# B&R Automation Studio project HISTest (part 7)

#### HMI_Alarm.st
```iecst
ACTION ActTimeSplit:
	(**********************************************************************************)
	(* TIME TRANS 'DT#YYYY-MM-DD-hh:mm:ss' >> 'YY-MM-DD, hh:mm' *)
	(**********************************************************************************)
	Timestamp.DTGetTime_0();

	Timestamp.Original := DT_TO_STRING(Timestamp.DTGetTime_0.DT1);
	Timestamp.Split.Day := MID(Timestamp.Original,8,6);
	Timestamp.Split.Time := MID(Timestamp.Original,5,15);

	Timestamp.Total := CONCAT(Timestamp.Split.Day, CONCAT(', ',Timestamp.Split.Time));
END_ACTION
ACTION ActSystem_Warning:

	IF EDGEPOS(PMS.SysBatProtect.Field.BSA_Alarm_OC) THEN
		IF HMI_Alarm.Warning[0].Count = 0 THEN
			HMI_Alarm.Warning[0].InitialTime 	:= Timestamp.Total;
			HMI_Alarm.Warning[0].RecentTime 	:= Timestamp.Total;
		ELSE
			HMI_Alarm.Warning[0].RecentTime 	:= Timestamp.Total;
		END_IF;
		HMI_Alarm.Warning[0].Count  := HMI_Alarm.Warning[0].Count + 1;
	END_IF;
	IF EDGEPOS(PMS.SysBatProtect.Field.BSA_Alarm_SOC_OV) THEN
		IF HMI_Alarm.Warning[1].Count = 0 THEN
			HMI_Alarm.Warning[1].InitialTime  	:= Timestamp.Total;
			HMI_Alarm.Warning[1].RecentTime 	:= Timestamp.Total;
		ELSE
			HMI_Alarm.Warning[1].InitialTime  	:= Timestamp.Total;
		END_IF;
		HMI_Alarm.Warning[1].Count  := HMI_Alarm.Warning[1].Count + 1;
	END_IF;
	IF EDGEPOS(PMS.SysBatProtect.Field.BSA_Alarm_SOC_UN) THEN
		IF HMI_Alarm.Warning[2].Count = 0 THEN
			HMI_Alarm.Warning[2].InitialTime  	:= Timestamp.Total;
			HMI_Alarm.Warning[2].RecentTime 	:= Timestamp.Total;
		ELSE
			HMI_Alarm.Warning[2].InitialTime  	:= Timestamp.Total;
		END_IF;
		HMI_Alarm.Warning[2].Count  := HMI_Alarm.Warning[2].Count + 1;
	END_IF;
	IF EDGEPOS(PMS.SysBatProtect.Field.BSA_Alarm_OV) THEN
		IF HMI_Alarm.Warning[3].Count = 0 THEN
			HMI_Alarm.Warning[3].InitialTime  	:= Timestamp.Total;
			HMI_Alarm.Warning[3].RecentTime 	:= Timestamp.Total;
		ELSE
			HMI_Alarm.Warning[3].InitialTime  	:= Timestamp.Total;
		END_IF;
		HMI_Alarm.Warning[3].Count  := HMI_Alarm.Warning[3].Count + 1;
	END_IF;
	IF EDGEPOS(PMS.SysBatProtect.Field.BSA_Alarm_UV) THEN
		IF HMI_Alarm.Warning[4].Count = 0 THEN
			HMI_Alarm.Warning[4].InitialTime  	:= Timestamp.Total;
			HMI_Alarm.Warning[4].RecentTime 	:= Timestamp.Total;
		ELSE
			HMI_Alarm.Warning[4].InitialTime  	:= Timestamp.Total;
		END_IF;
		HMI_Alarm.Warning[4].Count  := HMI_Alarm.Warning[4].Count + 1;
	END_IF;
	IF EDGEPOS(PMS.SysBatProtect.Field.BSA_Alarm_Cell_OV) THEN
		IF HMI_Alarm.Warning[5].Count = 0 THEN
			HMI_Alarm.Warning[5].InitialTime  	:= Timestamp.Total;
			HMI_Alarm.Warning[5].RecentTime 	:= Timestamp.Total;
		ELSE
			HMI_Alarm.Warning[5].InitialTime  	:= Timestamp.Total;
		END_IF;
		HMI_Alarm.Warning[5].Count  := HMI_Alarm.Warning[5].Count + 1;
	END_IF;
	IF EDGEPOS(PMS.SysBatProtect.Field.BSA_Alarm_Cell_UV) THEN
		IF HMI_Alarm.Warning[6].Count = 0 THEN
			HMI_Alarm.Warning[6].InitialTime  	:= Timestamp.Total;
			HMI_Alarm.Warning[6].RecentTime 	:= Timestamp.Total;
		ELSE
			HMI_Alarm.Warning[6].InitialTime  	:= Timestamp.Total;
		END_IF;
		HMI_Alarm.Warning[6].Count  := HMI_Alarm.Warning[6].Count + 1;
	END_IF;
	IF EDGEPOS(PMS.SysBatProtect.Field.BSA_Alarm_Cell_UnBalaV) THEN
		IF HMI_Alarm.Warning[7].Count = 0 THEN
			HMI_Alarm.Warning[7].InitialTime  	:= Timestamp.Total;
			HMI_Alarm.Warning[7].RecentTime 	:= Timestamp.Total;
		ELSE
			HMI_Alarm.Warning[7].InitialTime  	:= Timestamp.Total;
		END_IF;
		HMI_Alarm.Warning[7].Count  := HMI_Alarm.Warning[7].Count + 1;
	END_IF;
	IF EDGEPOS(PMS.SysBatProtect.Field.BSA_Alarm_Discharger_Cell_OT) THEN
		IF HMI_Alarm.Warning[8].Count = 0 THEN
			HMI_Alarm.Warning[8].InitialTime  	:= Timestamp.Total;
			HMI_Alarm.Warning[8].RecentTime 	:= Timestamp.Total;
		ELSE
			HMI_Alarm.Warning[8].InitialTime  	:= Timestamp.Total;
		END_IF;
		HMI_Alarm.Warning[8].Count  := HMI_Alarm.Warning[8].Count + 1;
	END_IF;
	IF EDGEPOS(PMS.SysBatProtect.Field.BSA_Alarm_Charger_Cell_OT) THEN
		IF HMI_Alarm.Warning[9].Count = 0 THEN
			HMI_Alarm.Warning[9].InitialTime  	:= Timestamp.Total;
			HMI_Alarm.Warning[9].RecentTime 	:= Timestamp.Total;
		ELSE
			HMI_Alarm.Warning[9].InitialTime  	:= Timestamp.Total;
		END_IF;
		HMI_Alarm.Warning[9].Count  := HMI_Alarm.Warning[9].Count + 1;
	END_IF;
	IF EDGEPOS(PMS.SysBatProtect.Field.BSA_Alarm_Discharger_Cell_UT) THEN
		IF HMI_Alarm.Warning[10].Count = 0 THEN
			HMI_Alarm.Warning[10].InitialTime  	:= Timestamp.Total;
			HMI_Alarm.Warning[10].RecentTime 	:= Timestamp.Total;
		ELSE
			HMI_Alarm.Warning[10].InitialTime  	:= Timestamp.Total;
		END_IF;
		HMI_Alarm.Warning[10].Count 	:= HMI_Alarm.Warning[10].Count + 1;
	END_IF;
	IF EDGEPOS(PMS.SysBatProtect.Field.BSA_Alarm_Charger_Cell_UT) THEN
		IF HMI_Alarm.Warning[11].Count = 0 THEN
			HMI_Alarm.Warning[11].InitialTime  	:= Timestamp.Total;
			HMI_Alarm.Warning[11].RecentTime 	:= Timestamp.Total;
		ELSE
			HMI_Alarm.Warning[11].InitialTime  	:= Timestamp.Total;
		END_IF;
		HMI_Alarm.Warning[11].Count 	:= HMI_Alarm.Warning[11].Count + 1;
	END_IF;
	IF EDGEPOS(PMS.SysBatProtect.Field.BSA_Alarm_Cell_UnBalaT) THEN
		IF HMI_Alarm.Warning[12].Count = 0 THEN
			HMI_Alarm.Warning[12].InitialTime  	:= Timestamp.Total;
			HMI_Alarm.Warning[12].RecentTime 	:= Timestamp.Total;
		ELSE
			HMI_Alarm.Warning[12].InitialTime  	:= Timestamp.Total;
		END_IF;
		HMI_Alarm.Warning[12].Count 	:= HMI_Alarm.Warning[12].Count + 1;
	END_IF;

END_ACTION
ACTION ActSystem_Fault: //
	IF EDGEPOS(PMS.SysBatProtect.Field.BSA_Fault_OC) THEN
		IF HMI_Alarm.Fault[0].Count = 0 THEN
			HMI_Alarm.Fault[0].InitialTime 	:= Timestamp.Total;
			HMI_Alarm.Fault[0].RecentTime 	:= Timestamp.Total;
		ELSE
			HMI_Alarm.Fault[0].RecentTime 	:= Timestamp.Total;
		END_IF;
		HMI_Alarm.Fault[0].Count  := HMI_Alarm.Fault[0].Count + 1;
	END_IF;
	IF EDGEPOS(PMS.SysBatProtect.Field.BSA_Fault_SOC_OV) THEN
		IF HMI_Alarm.Fault[1].Count = 0 THEN
			HMI_Alarm.Fault[1].InitialTime  	:= Timestamp.Total;
			HMI_Alarm.Fault[1].RecentTime 	:= Timestamp.Total;
		ELSE
			HMI_Alarm.Fault[1].InitialTime  	:= Timestamp.Total;
		END_IF;
		HMI_Alarm.Fault[1].Count  := HMI_Alarm.Fault[1].Count + 1;
	END_IF;
	IF EDGEPOS(PMS.SysBatProtect.Field.BSA_Fault_SOC_UN) THEN
		IF HMI_Alarm.Fault[2].Count = 0 THEN
			HMI_Alarm.Fault[2].InitialTime  	:= Timestamp.Total;
			HMI_Alarm.Fault[2].RecentTime 	:= Timestamp.Total;
		ELSE
			HMI_Alarm.Fault[2].InitialTime  	:= Timestamp.Total;
		END_IF;
		HMI_Alarm.Fault[2].Count  := HMI_Alarm.Fault[2].Count + 1;
	END_IF;
	IF EDGEPOS(PMS.SysBatProtect.Field.BSA_Fault_OV) THEN
		IF HMI_Alarm.Fault[3].Count = 0 THEN
			HMI_Alarm.Fault[3].InitialTime  	:= Timestamp.Total;
			HMI_Alarm.Fault[3].RecentTime 	:= Timestamp.Total;
		ELSE
			HMI_Alarm.Fault[3].InitialTime  	:= Timestamp.Total;
		END_IF;
		HMI_Alarm.Fault[3].Count  := HMI_Alarm.Fault[3].Count + 1;
	END_IF;
	IF EDGEPOS(PMS.SysBatProtect.Field.BSA_Fault_UV) THEN
		IF HMI_Alarm.Fault[4].Count = 0 THEN
			HMI_Alarm.Fault[4].InitialTime  	:= Timestamp.Total;
			HMI_Alarm.Fault[4].RecentTime 	:= Timestamp.Total;
		ELSE
			HMI_Alarm.Fault[4].InitialTime  	:= Timestamp.Total;
		END_IF;
		HMI_Alarm.Fault[4].Count  := HMI_Alarm.Fault[4].Count + 1;
	END_IF;
	IF EDGEPOS(PMS.SysBatProtect.Field.BSA_Fault_Cell_OV) THEN
		IF HMI_Alarm.Fault[5].Count = 0 THEN
			HMI_Alarm.Fault[5].InitialTime  	:= Timestamp.Total;
			HMI_Alarm.Fault[5].RecentTime 	:= Timestamp.Total;
		ELSE
			HMI_Alarm.Fault[5].InitialTime  	:= Timestamp.Total;
		END_IF;
		HMI_Alarm.Fault[5].Count  := HMI_Alarm.Fault[5].Count + 1;
	END_IF;
	IF EDGEPOS(PMS.SysBatProtect.Field.BSA_Fault_Cell_UV) THEN
		IF HMI_Alarm.Fault[6].Count = 0 THEN
			HMI_Alarm.Fault[6].InitialTime  	:= Timestamp.Total;
			HMI_Alarm.Fault[6].RecentTime 	:= Timestamp.Total;
		ELSE
			HMI_Alarm.Fault[6].InitialTime  	:= Timestamp.Total;
		END_IF;
		HMI_Alarm.Fault[6].Count  := HMI_Alarm.Fault[6].Count + 1;
	END_IF;
	IF EDGEPOS(PMS.SysBatProtect.Field.BSA_Fault_Cell_UnBalaV) THEN
		IF HMI_Alarm.Fault[7].Count = 0 THEN
			HMI_Alarm.Fault[7].InitialTime  	:= Timestamp.Total;
			HMI_Alarm.Fault[7].RecentTime 	:= Timestamp.Total;
		ELSE
			HMI_Alarm.Fault[7].InitialTime  	:= Timestamp.Total;
		END_IF;
		HMI_Alarm.Fault[7].Count  := HMI_Alarm.Fault[7].Count + 1;
	END_IF;
	IF EDGEPOS(PMS.SysBatProtect.Field.BSA_Fault_Discharger_Cell_OT) THEN
		IF HMI_Alarm.Fault[8].Count = 0 THEN
			HMI_Alarm.Fault[8].InitialTime  	:= Timestamp.Total;
			HMI_Alarm.Fault[8].RecentTime 	:= Timestamp.Total;
		ELSE
			HMI_Alarm.Fault[8].InitialTime  	:= Timestamp.Total;
		END_IF;
		HMI_Alarm.Fault[8].Count  := HMI_Alarm.Fault[8].Count + 1;
	END_IF;
	IF EDGEPOS(PMS.SysBatProtect.Field.BSA_Fault_Charger_Cell_OT) THEN
		IF HMI_Alarm.Fault[9].Count = 0 THEN
			HMI_Alarm.Fault[9].InitialTime  	:= Timestamp.Total;
			HMI_Alarm.Fault[9].RecentTime 	:= Timestamp.Total;
		ELSE
			HMI_Alarm.Fault[9].InitialTime  	:= Timestamp.Total;
		END_IF;
		HMI_Alarm.Fault[9].Count  := HMI_Alarm.Fault[9].Count + 1;
	END_IF;
	IF EDGEPOS(PMS.SysBatProtect.Field.BSA_Fault_Discharger_Cell_UT) THEN
		IF HMI_Alarm.Fault[10].Count = 0 THEN
			HMI_Alarm.Fault[10].InitialTime  	:= Timestamp.Total;
			HMI_Alarm.Fault[10].RecentTime 	:= Timestamp.Total;
		ELSE
			HMI_Alarm.Fault[10].InitialTime  	:= Timestamp.Total;
		END_IF;
		HMI_Alarm.Fault[10].Count 	:= HMI_Alarm.Fault[10].Count + 1;
	END_IF;
	IF EDGEPOS(PMS.SysBatProtect.Field.BSA_Fault_Charger_Cell_UT) THEN
		IF HMI_Alarm.Fault[11].Count = 0 THEN
			HMI_Alarm.Fault[11].InitialTime  	:= Timestamp.Total;
			HMI_Alarm.Fault[11].RecentTime 	:= Timestamp.Total;
		ELSE
			HMI_Alarm.Fault[11].InitialTime  	:= Timestamp.Total;
		END_IF;
		HMI_Alarm.Fault[11].Count 	:= HMI_Alarm.Fault[11].Count + 1;
	END_IF;
	IF EDGEPOS(PMS.SysBatProtect.Field.BSA_Fault_Cell_UnBalaT) THEN
		IF HMI_Alarm.Fault[12].Count = 0 THEN
			HMI_Alarm.Fault[12].InitialTime  	:= Timestamp.Total;
			HMI_Alarm.Fault[12].RecentTime 	:= Timestamp.Total;
		ELSE
			HMI_Alarm.Fault[12].InitialTime  	:= Timestamp.Total;
		END_IF;
		HMI_Alarm.Fault[12].Count 	:= HMI_Alarm.Fault[12].Count + 1;
	END_IF;
END_ACTION
ACTION ActSystem_Protect:

	IF EDGEPOS(PMS.SysBatProtect.Field.BSA_Prtct_OC) THEN

		IF HMI_Alarm.Protect[0].Count = 0 THEN
			HMI_Alarm.Protect[0].InitialTime 	:= Timestamp.Total;
			HMI_Alarm.Protect[0].RecentTime 	:= Timestamp.Total;
		ELSE
			HMI_Alarm.Protect[0].RecentTime 	:= Timestamp.Total;
		END_IF;
		HMI_Alarm.Protect[0].Count  := HMI_Alarm.Protect[0].Count + 1;
	END_IF;
	IF EDGEPOS(PMS.SysBatProtect.Field.BSA_Prtct_SOC_OV) THEN

		IF HMI_Alarm.Protect[1].Count = 0 THEN
			HMI_Alarm.Protect[1].InitialTime  	:= Timestamp.Total;
			HMI_Alarm.Protect[1].RecentTime 	:= Timestamp.Total;
		ELSE
			HMI_Alarm.Protect[1].RecentTime  	:= Timestamp.Total;
		END_IF;
		HMI_Alarm.Protect[1].Count  := HMI_Alarm.Protect[1].Count + 1;
	END_IF;
	IF EDGEPOS(PMS.SysBatProtect.Field.BSA_Prtct_SOC_UN) THEN

		IF HMI_Alarm.Protect[2].Count = 0 THEN
			HMI_Alarm.Protect[2].InitialTime  	:= Timestamp.Total;
			HMI_Alarm.Protect[2].RecentTime 	:= Timestamp.Total;
		ELSE
			HMI_Alarm.Protect[2].RecentTime  	:= Timestamp.Total;
		END_IF;
		HMI_Alarm.Protect[2].Count  := HMI_Alarm.Protect[2].Count + 1;
	END_IF;
	IF EDGEPOS(PMS.SysBatProtect.Field.BSA_Prtct_OV) THEN

		IF HMI_Alarm.Protect[3].Count = 0 THEN
			HMI_Alarm.Protect[3].InitialTime  	:= Timestamp.Total;
			HMI_Alarm.Protect[3].RecentTime 	:= Timestamp.Total;
		ELSE
			HMI_Alarm.Protect[3].RecentTime  	:= Timestamp.Total;
		END_IF;
		HMI_Alarm.Protect[3].Count  := HMI_Alarm.Protect[3].Count + 1;
	END_IF;
	IF EDGEPOS(PMS.SysBatProtect.Field.BSA_Prtct_UV) THEN

		IF HMI_Alarm.Protect[4].Count = 0 THEN
			HMI_Alarm.Protect[4].InitialTime  	:= Timestamp.Total;
			HMI_Alarm.Protect[4].RecentTime 	:= Timestamp.Total;
		ELSE
			HMI_Alarm.Protect[4].RecentTime  	:= Timestamp.Total;
		END_IF;
		HMI_Alarm.Protect[4].Count  := HMI_Alarm.Protect[4].Count + 1;
	END_IF;
	IF EDGEPOS(PMS.SysBatProtect.Field.BSA_Prtct_Cell_OV) THEN

		IF HMI_Alarm.Protect[5].Count = 0 THEN
			HMI_Alarm.Protect[5].InitialTime  	:= Timestamp.Total;
			HMI_Alarm.Protect[5].RecentTime 	:= Timestamp.Total;
		ELSE
			HMI_Alarm.Protect[5].RecentTime  	:= Timestamp.Total;
		END_IF;
		HMI_Alarm.Protect[5].Count  := HMI_Alarm.Protect[5].Count + 1;
	END_IF;
	IF EDGEPOS(PMS.SysBatProtect.Field.BSA_Prtct_Cell_UV) THEN

		IF HMI_Alarm.Protect[6].Count = 0 THEN
			HMI_Alarm.Protect[6].InitialTime  	:= Timestamp.Total;
			HMI_Alarm.Protect[6].RecentTime 	:= Timestamp.Total;
		ELSE
			HMI_Alarm.Protect[6].RecentTime  	:= Timestamp.Total;
		END_IF;
		HMI_Alarm.Protect[6].Count  := HMI_Alarm.Protect[6].Count + 1;
	END_IF;
	IF EDGEPOS(PMS.SysBatProtect.Field.BSA_Prtct_Cell_UnBalaV) THEN

		IF HMI_Alarm.Protect[7].Count = 0 THEN
			HMI_Alarm.Protect[7].InitialTime  	:= Timestamp.Total;
			HMI_Alarm.Protect[7].RecentTime 	:= Timestamp.Total;
		ELSE
			HMI_Alarm.Protect[7].RecentTime  	:= Timestamp.Total;
		END_IF;
		HMI_Alarm.Protect[7].Count  := HMI_Alarm.Protect[7].Count + 1;
	END_IF;
	IF EDGEPOS(PMS.SysBatProtect.Field.BSA_Prtct_Discharger_Cell_OT) THEN

		IF HMI_Alarm.Protect[8].Count = 0 THEN
			HMI_Alarm.Protect[8].InitialTime  	:= Timestamp.Total;
			HMI_Alarm.Protect[8].RecentTime 	:= Timestamp.Total;
		ELSE
			HMI_Alarm.Protect[8].RecentTime  	:= Timestamp.Total;
		END_IF;
		HMI_Alarm.Protect[8].Count  := HMI_Alarm.Protect[8].Count + 1;
	END_IF;
	IF EDGEPOS(PMS.SysBatProtect.Field.BSA_Prtct_Charger_Cell_OT) THEN

		IF HMI_Alarm.Protect[9].Count = 0 THEN
			HMI_Alarm.Protect[9].InitialTime  	:= Timestamp.Total;
			HMI_Alarm.Protect[9].RecentTime 	:= Timestamp.Total;
		ELSE
			HMI_Alarm.Protect[9].RecentTime  	:= Timestamp.Total;
		END_IF;
		HMI_Alarm.Protect[9].Count  := HMI_Alarm.Protect[9].Count + 1;
	END_IF;
	IF EDGEPOS(PMS.SysBatProtect.Field.BSA_Prtct_Discharger_Cell_UT) THEN

		IF HMI_Alarm.Protect[10].Count = 0 THEN
			HMI_Alarm.Protect[10].InitialTime  	:= Timestamp.Total;
			HMI_Alarm.Protect[10].RecentTime 	:= Timestamp.Total;
		ELSE
			HMI_Alarm.Protect[10].RecentTime  	:= Timestamp.Total;
		END_IF;
		HMI_Alarm.Protect[10].Count 	:= HMI_Alarm.Protect[10].Count + 1;
	END_IF;
	IF EDGEPOS(PMS.SysBatProtect.Field.BSA_Prtct_Charger_Cell_UT) THEN

		IF HMI_Alarm.Protect[11].Count = 0 THEN
			HMI_Alarm.Protect[11].InitialTime  	:= Timestamp.Total;
			HMI_Alarm.Protect[11].RecentTime 	:= Timestamp.Total;
		ELSE
			HMI_Alarm.Protect[11].RecentTime  	:= Timestamp.Total;
		END_IF;
		HMI_Alarm.Protect[11].Count 	:= HMI_Alarm.Protect[11].Count + 1;
	END_IF;
	IF EDGEPOS(PMS.SysBatProtect.Field.BSA_Prtct_Cell_UnBalaT) THEN

		IF HMI_Alarm.Protect[12].Count = 0 THEN
			HMI_Alarm.Protect[12].InitialTime  	:= Timestamp.Total;
			HMI_Alarm.Protect[12].RecentTime 	:= Timestamp.Total;
		ELSE
			HMI_Alarm.Protect[12].RecentTime  	:= Timestamp.Total;
		END_IF;
		HMI_Alarm.Protect[12].Count 	:= HMI_Alarm.Protect[12].Count + 1;
	END_IF;
	IF EDGEPOS(PMS.SysBatProtect.Field.BSA_Prtct_RelayWelding) THEN

		IF HMI_Alarm.Protect[13].Count = 0 THEN
			HMI_Alarm.Protect[13].InitialTime  	:= Timestamp.Total;
			HMI_Alarm.Protect[13].RecentTime 	:= Timestamp.Total;
		ELSE
			HMI_Alarm.Protect[13].RecentTime  	:= Timestamp.Total;
		END_IF;
		HMI_Alarm.Protect[13].Count 	:= HMI_Alarm.Protect[13].Count + 1;
	END_IF;
	IF EDGEPOS(PMS.SysBatProtect.Field.BSA_Prtct_InternalCOM) THEN

		IF HMI_Alarm.Protect[14].Count = 0 THEN
			HMI_Alarm.Protect[14].InitialTime  	:= Timestamp.Total;
			HMI_Alarm.Protect[14].RecentTime 	:= Timestamp.Total;
		ELSE
			HMI_Alarm.Protect[14].RecentTime  	:= Timestamp.Total;
		END_IF;
		HMI_Alarm.Protect[14].Count 	:= HMI_Alarm.Protect[14].Count + 1;
	END_IF;
	IF EDGEPOS(PMS.SysBatProtect.Field.BSA_Prtct_ExternalCOM) THEN

		IF HMI_Alarm.Protect[15].Count = 0 THEN
			HMI_Alarm.Protect[15].InitialTime  	:= Timestamp.Total;
			HMI_Alarm.Protect[15].RecentTime 	:= Timestamp.Total;
		ELSE
			HMI_Alarm.Protect[15].RecentTime  	:= Timestamp.Total;
		END_IF;
		HMI_Alarm.Protect[15].Count 	:= HMI_Alarm.Protect[15].Count + 1;
	END_IF;
//	IF EDGEPOS(PMS.SysBatProtect.Field.BSA_Prtct_CT_COM_Err) THEN
//
//		IF HMI_Alarm.Protect[16].Count = 0 THEN
//			HMI_Alarm.Protect[16].InitialTime  	:= Timestamp.Total;
//			HMI_Alarm.Protect[16].RecentTime 	:= Timestamp.Total;
//		ELSE
//			HMI_Alarm.Protect[16].InitialTime  	:= Timestamp.Total;
//		END_IF;
//		HMI_Alarm.Protect[16].Count 	:= HMI_Alarm.Protect[16].Count + 1;
//	END_IF;
	IF EDGEPOS(PMS.SysBatProtect.Field.BSA_Prtct_WaterLeak) THEN

		IF HMI_Alarm.Protect[17].Count = 0 THEN
			HMI_Alarm.Protect[17].InitialTime  	:= Timestamp.Total;
			HMI_Alarm.Protect[17].RecentTime 	:= Timestamp.Total;
		ELSE
			HMI_Alarm.Protect[17].RecentTime  	:= Timestamp.Total;
		END_IF;
		HMI_Alarm.Protect[17].Count 	:= HMI_Alarm.Protect[17].Count + 1;
	END_IF;
//	IF EDGEPOS(PMS.SysBatProtect.Field.BSA_Prtct_EMS_SW_Err) THEN
//
//		IF HMI_Alarm.Protect[18].Count = 0 THEN
//			HMI_Alarm.Protect[18].InitialTime  	:= Timestamp.Total;
//			HMI_Alarm.Protect[18].RecentTime 	:= Timestamp.Total;
//		ELSE
//			HMI_Alarm.Protect[18].InitialTime  	:= Timestamp.Total;
//		END_IF;
//		HMI_Alarm.Protect[18].Count 	:= HMI_Alarm.Protect[18].Count + 1;
//	END_IF;

	IF NOT(HMI.DialogBox.Protect_Trigger) THEN
		FOR LoopNum := 0 TO 18 DO
			IF HMI_Alarm.Protect[LoopNum].Count > 0 THEN
				HMI.DialogBox.Protect_Trigger 	:= TRUE;
				HMI.DialogBox.ProtectName		:=	HMI_Alarm.Protect[LoopNum].Name;
				EXIT;
			END_IF;
		END_FOR;
	END_IF;

END_ACTION

ACTION ActSystem_AlarmTab:
	CASE HMI.AlarmTableIndex OF
		vkWarning:
			memcpy(ADR(HMI.SubBMS_AlarmTable), ADR(HMI_Alarm.Warning), SIZEOF(HMI_Alarm.Warning));

		vkFault:
			memcpy(ADR(HMI.SubBMS_AlarmTable), ADR(HMI_Alarm.Fault), SIZEOF(HMI_Alarm.Fault));

		vkProtect:
			memcpy(ADR(HMI.SubBMS_AlarmTable), ADR(HMI_Alarm.Protect), SIZEOF(HMI_Alarm.Protect));

	END_CASE;
END_ACTION
```

#### HMI_Common.st
```iecst
ACTION ActTrendData:
	HMI.TrendData.Voltage	:= UINT_TO_REAL(PMS.SysBatCal.Field.BSA_Volt_Total);
	HMI.TrendData.Current	:= UINT_TO_REAL(PMS.SysBatCal.Field.BSA_Curr_Total);
END_ACTION
```

#### HMI_Event.st
```iecst
ACTION ActLOGIN	:
	IF NOT(HMI.AdminLogin.Input_Button = '') THEN
		IF (HMI.AdminLogin.Input_Button = 'E') THEN
			IF NOT(LEN(HMI.AdminLogin.Password_Internal) = 0) THEN
				HMI.AdminLogin.Password_Internal 	:= LEFT(HMI.AdminLogin.Password_Internal,LEN(HMI.AdminLogin.Password_Internal)-1);
				HMI.AdminLogin.Password_External 	:= LEFT(HMI.AdminLogin.Password_External,LEN(HMI.AdminLogin.Password_External)-1);
			END_IF;
		ELSIF (HMI.AdminLogin.Input_Button = 'L') THEN
			IF HMI.AdminLogin.Password_Internal = PASSWORD THEN
				HMI.AdminLogin.Authority 		:= ADMIN;
				HMI.AdminLogin.Password_Internal:= '';
				HMI.AdminLogin.Password_External:= '';
			END_IF;
		ELSE
			HMI.AdminLogin.Password_Internal 	:= CONCAT(HMI.AdminLogin.Password_Internal,HMI.AdminLogin.Input_Button);
			HMI.AdminLogin.Password_External 	:= CONCAT(HMI.AdminLogin.Password_External,'*');
		END_IF;
		HMI.AdminLogin.Input_Button 		:= '';
	END_IF;
END_ACTION

ACTION ActDeviceReset:
	IF (HMI.AdminDeviceReset) THEN

		StateMa := vkSYSTEM_PROTECT_CHECK;
		FOR LoopNum := 0 TO 18 DO
			HMI_Alarm.Fault[LoopNum].InitialTime		:=	'';
			HMI_Alarm.Fault[LoopNum].RecentTime			:=	'';
			HMI_Alarm.Fault[LoopNum].ClearTime			:=	'';
			HMI_Alarm.Fault[LoopNum].Count				:=	0;
			HMI_Alarm.Warning[LoopNum].InitialTime		:=	'';
			HMI_Alarm.Warning[LoopNum].RecentTime		:=	'';
			HMI_Alarm.Warning[LoopNum].ClearTime		:=	'';
			HMI_Alarm.Warning[LoopNum].Count			:=	0;
			HMI_Alarm.Protect[LoopNum].InitialTime		:=	'';
			HMI_Alarm.Protect[LoopNum].RecentTime		:=	'';
			HMI_Alarm.Protect[LoopNum].ClearTime		:=	'';
			HMI_Alarm.Protect[LoopNum].Count			:=	0;

		END_FOR;

		HMI.DialogBox.Protect_Trigger := FALSE;
		HMI.AdminDeviceReset := FALSE;

	END_IF;
END_ACTION
```

#### HMI_DeviceLoading.st - not listed in the package file held
```iecst
ACTION ActDeviceloading:

	TON_0();

	CASE HMI.DeviceLoading.DeviceLoadingStep OF
		0:
			HMI.DeviceLoading.RackLoading := 0;

		1:// 통신확인

			TON_0.IN							:= TRUE;

			HMI.DeviceLoading.Trigger 			:= FALSE;

			HMI.DeviceLoading.DeviceLoadingStep := 2;
			HMI.DeviceLoading.RackLoading 		:= 1;

		2:// Rack 갯수 설정

			HMI.DeviceLoading.RackLoading := 2;

			IF HMI.DeviceLoading.SetRackNum <> 0 THEN

				HMI.DeviceLoading.DeviceLoading_Max := HMI.DeviceLoading.DeviceLoadingStep + HMI.DeviceLoading.SetRackNum;

				HMI.DeviceLoading.DeviceLoadingStep := 3;

			ELSE
				HMI.DeviceLoading.Trigger := TRUE;
			END_IF;

		3: // Rack 정보 확인

			FOR LoopCount := 0 TO (RACK_MAXNUM_MINUS_1) DO //RACK_NUMBER_MINUS_1 DO
				IF SubBMS_Calculator.BSA[LoopCount].Rack_State.Field.BSA_Divice_Status <> 0 THEN
					IF NOT(HMI.RackEnable[LoopCount]) THEN
						HMI.DeviceLoading.RackLoading 	:= HMI.DeviceLoading.RackLoading + 1;
						HMI.RackEnable[LoopCount]		:= TRUE;
					END_IF;

				END_IF;
			END_FOR;

			IF HMI.DeviceLoading.RackLoading = (HMI.DeviceLoading.DeviceLoading_Max)  THEN
				HMI.DeviceLoading.DeviceLoadingStep := 4;

				TON_0.IN							:= FALSE;

				HMI.DialogBox.Protect_Trigger 		:= FALSE;

				HMI.AlarmTableIndex := vkProtect;

			END_IF;
		4: // PROTECT 이력확인
			FOR i  := 0 TO 27 DO
				IF HMI_Alarm.Protect[i].Internal_Count <> 0  THEN
					HMI.DialogBox.Protect_Trigger 	:= TRUE;
					Sys.ProtectSig					:= TRUE;
					HMI.DialogBox.ProtectName		:= HMI_Alarm.Protect[i].Name;
					HMI.DialogBox.ProtectNum		:= HMI_Alarm.Protect[i].Location;
				END_IF;
			END_FOR;

			HMI.DeviceLoading.DeviceLoadingStep := 5;
			HMI.AlarmTableIndex := vkWarning;

		5: // Device Loading Done

			Sys.DeviceloadingDone := TRUE;

	END_CASE;

	IF TON_0.Q THEN
		HMI.DialogBox.LoadingError_Trigger := TRUE;
	END_IF;
END_ACTION
```

### Program Logical/Source/HMI/HMI_DeviceLoading (IEC)

#### Variables.var
```iecst
VAR
	LoopCount : INT;
	New_Variable : USINT;
	TON_0 : TON;
END_VAR
```

#### Main.st
```iecst
PROGRAM _INIT
	(* Insert code here *)

	HMI.DeviceLoading.DeviceLoadingStep := 0;
	HMI.DeviceLoading.SetRackNum		:= 0;
	HMI.DeviceLoading.RackLoading		:= 0;

	TON_0.PT := T#30s;

END_PROGRAM

PROGRAM _CYCLIC
	(* Insert code here *)
	TON_0();

	CASE HMI.DeviceLoading.DeviceLoadingStep OF
		0:
			HMI.DeviceLoading.RackLoading := 0;

		1:// 통신확인

			TON_0.IN							:= TRUE;

			HMI.DeviceLoading.Trigger 			:= FALSE;

			HMI.DeviceLoading.DeviceLoadingStep := 2;
			HMI.DeviceLoading.RackLoading 		:= 1;

		2:// Rack 갯수 설정

			HMI.DeviceLoading.RackLoading := 2;

			IF HMI.DeviceLoading.SetRackNum <> 0 THEN

				HMI.DeviceLoading.DeviceLoading_Max := HMI.DeviceLoading.DeviceLoadingStep + HMI.DeviceLoading.SetRackNum;

				HMI.DeviceLoading.DeviceLoadingStep := 3;

			ELSE
				HMI.DeviceLoading.Trigger := TRUE;
			END_IF;

		3: // Rack 정보 확인

			FOR LoopCount := 0 TO (RACK_MAXNUM_MINUS_1) DO //RACK_NUMBER_MINUS_1 DO
				IF SubBMS_Calculator.BSA[LoopCount].Rack_State.Field.BSA_Divice_Status <> 0 THEN
					IF NOT(HMI.RackEnable[LoopCount]) THEN
						HMI.DeviceLoading.RackLoading 	:= HMI.DeviceLoading.RackLoading + 1;
						HMI.RackEnable[LoopCount]		:= TRUE;
					END_IF;

				END_IF;
			END_FOR;

			IF HMI.DeviceLoading.RackLoading = (HMI.DeviceLoading.DeviceLoading_Max)  THEN
				HMI.DeviceLoading.DeviceLoadingStep := 4;
				TON_0.IN							:= FALSE;
			END_IF;
		4:

			HMI.Step := vkSYSTEM;
			HMI.DeviceLoading.DeviceLoadingStep := 5;

		5: // Device Loading Done

			FOR LoopCount := 0 TO (RACK_MAXNUM_MINUS_1) DO //RACK_NUMBER_MINUS_1 DO

				IF SubBMS_Calculator.BSA[LoopCount].Rack_State.Field.BSA_Divice_Status <> 0 THEN
					IF NOT(HMI.RackEnable[LoopCount]) THEN
						HMI.RackEnable[LoopCount]		:= TRUE;
					END_IF;
				ELSE
					IF (HMI.RackEnable[LoopCount]) THEN
						HMI.RackEnable[LoopCount]		:= FALSE;
					END_IF;
				END_IF;
			END_FOR;

	END_CASE;

	IF TON_0.Q THEN
		HMI.DialogBox.LoadingError_Trigger := TRUE;
	END_IF;

END_PROGRAM

PROGRAM _EXIT
	(* Insert code here *)

END_PROGRAM
```

Listed in the project but not available here: Logical/Libraries, Logical/Document, Logical/ArCan/J1939, Logical/MbTCP, Logical/Source/gStruct/PMS_TCP.typ, Logical/Source/SubBMS_CAN/CANRxSubBMS/ArCanReceive.typ, Logical/Source/SubBMS_CAN/CANTxSubBMS/ArCanSend.typ, Logical/Source/SubBMS_CAN/CANTxSubBMS/ArCanSend.var, Logical/Source/SubBMS_CAN/CANTxSubBMS/CanSend.st, Logical/Source/PMS_CAN/CANTxPMS/ArCanSend.typ, Logical/Source/PMS_CAN/CANTxPMS/ArCanSend.var, Logical/Source/PMS_CAN/CANTxPMS/Action.st, Logical/Source/PMS_CAN/CANRxPMS/ArCanReceive.typ, Logical/Source/PMS_CAN/CANRxPMS/ArCanReceive.var, Logical/Source/PMS_CAN/CANRxPMS/Action.st, Logical/Source/PMS_CAN/PMS_Calculator/Types.typ, Logical/Source/HMI/HMI_DataParsing/Types.typ
